TYPE "TExtEncoder_Sts"
VERSION : 0.1
// Block: TExtEncoder_Sts
   STRUCT
      AlarmPresence : Bool;
      Standstill : Bool;
      InOperation : Bool;
      HomingDone : Bool;
      ActualPosition : LReal;
   END_STRUCT;

END_TYPE
